Omron CX-Programmer project 新工程 (CX-Programmer 9.73)

# PLC 新PLC1: CPM1(CPM1A) CPU30

## Global symbols (name address type ; comment)
0.00 BOOL  ; 启动按钮
0.01 BOOL  ; 0号机停按钮
0.02 BOOL  ; 1号机停按钮
0.03 BOOL  ; 2号电停按钮
10.00 BOOL  ; 0号电机
10.01 BOOL  ; 1号电机
10.02 BOOL  ; 2号电机
200.00 BOOL  ; 0号电机运行
200.01 BOOL  ; 1号电机运行
200.02 BOOL  ; 2号电机运行
TIM000 BOOL  ; 1号电机延时5秒启动
TIM001 BOOL  ; 1号机延5秒启动
TIM002 BOOL  ; 2号机延5秒启动
TIM003 BOOL  ; 1号电机延时停
TIM004 BOOL  ; 0号电机延时停
TIM005 BOOL  ; 1号电机延时停

## Program 新程序1 (no task)
; 简介： / 这个PLC程序实现了一个三电机延时启停控制系统，适用于生产线上的输送带系统，驱动进料段、主输送段和出料段的三台电机。系统通过启动按钮触发整个流程，依次启动三台电机，并通过各自的停止按钮控制关闭。顺序启动设计避免了三台电机同时启动带来的电流冲击，停止时部分电机需延时关闭以保护设备。 / 采用设备： / 系统包含操作面板上的启动按钮、0号机停按钮、1号机停按钮和2号机停按钮。执行器包括0号电机、1号电机和2号电机，分别驱动输送带的进料段、主输送段和出料段。 / 系统流程： / 系统通过启动按钮启动整个流程，首先激活0号电机驱动进料段开始工作。此时，0号电机运行置位，反映进料段的运行状态，且其状态必须始终与0号电机的实际启停保持一致，以确保系统监控的准确性。 / 0号电机运行时，1号电机延时5秒启动开始计时5秒。计时完成后，1号电机启动，驱动主输送段，保证物料平稳过渡。 / 1号电机运行时，2号电机延时5秒启动开始计时5秒。计时完成后，2号电机启动，驱动出料段，确保物料顺利流动。 / 1号电机和2号电机的运行状态分别反映主输送段和出料段的状况。 / 在运行过程中，操作员可通过0号机停按钮、1号机停按钮和2号机停按钮分别控制三段电机的停止。 / 值得注意的是，启动按钮与这些停止按钮不能同时按下，否则可能导致0号电机的状态异常，例如意外启动或停止，影响物料流动的稳定性。 / 按下0号机停按钮时，0号电机延时停开始计时5秒，之后关闭0号电机，确保进料段物料清空。 / 按下1号机停按钮时，1号电机延时停开始计时5秒，之后关闭1号电机，保证主输送段物料平稳过渡。 / 而2号机停按钮按下时，2号电机直接停止。

### Section 段1

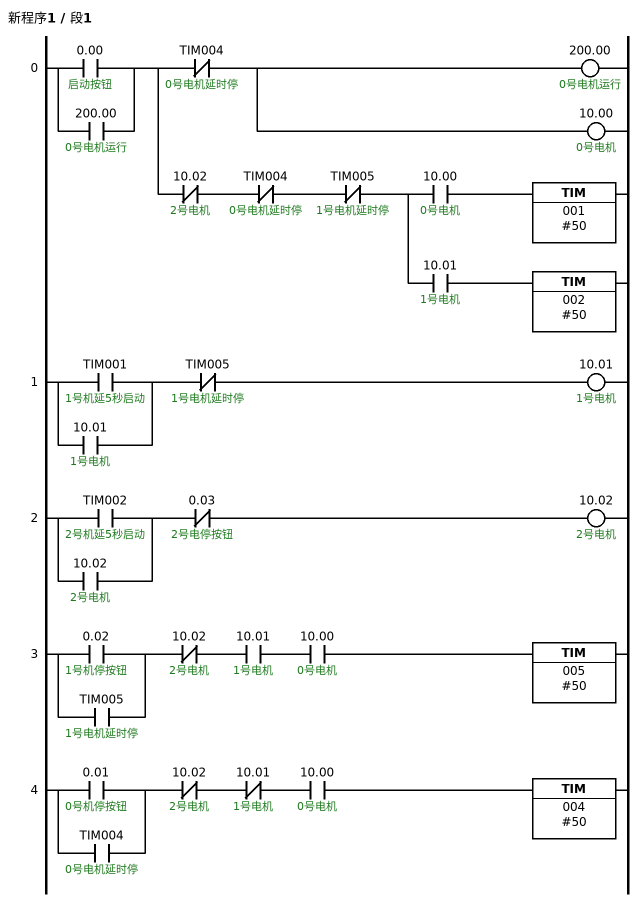
; rung 0
LD 0.00  ; 启动按钮
OR 200.00  ; 0号电机运行
OUT TR0
ANDNOT TIM004  ; 0号电机延时停
OUT 200.00  ; 0号电机运行
OUT 10.00  ; 0号电机
LD TR0
ANDNOT 10.02  ; 2号电机
ANDNOT TIM004  ; 0号电机延时停
ANDNOT TIM005  ; 1号电机延时停
OUT TR0
AND 10.00  ; 0号电机
TIM 001 #50
LD TR0
AND 10.01  ; 1号电机
TIM 002 #50
; rung 1
LD TIM001  ; 1号机延5秒启动
OR 10.01  ; 1号电机
ANDNOT TIM005  ; 1号电机延时停
OUT 10.01  ; 1号电机
; rung 2
LD TIM002  ; 2号机延5秒启动
OR 10.02  ; 2号电机
ANDNOT 0.03  ; 2号电停按钮
OUT 10.02  ; 2号电机
; rung 3
LD 0.02  ; 1号机停按钮
OR TIM005  ; 1号电机延时停
ANDNOT 10.02  ; 2号电机
AND 10.01  ; 1号电机
AND 10.00  ; 0号电机
TIM 005 #50
; rung 4
LD 0.01  ; 0号机停按钮
OR TIM004  ; 0号电机延时停
ANDNOT 10.02  ; 2号电机
ANDNOT 10.01  ; 1号电机
AND 10.00  ; 0号电机
TIM 004 #50
; rung 5
END(01)